FUNCTION_BLOCK TESTE
  (* Standard: 61499-2 *)
  (* Version 11-01-12, GASR *)
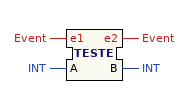
  EVENT_INPUT
    e1;
  END_EVENT
  EVENT_OUTPUT
    e2;
  END_EVENT
  VAR_INPUT
    A : INT;
  END_VAR
  VAR_OUTPUT
    B : INT;
  END_VAR
  EC_STATES
    START;
  END_STATES
END_FUNCTION_BLOCK
